// SIMATIC S7-200 SMART project (STEP 7-Micro/WIN SMART), CPU SR40

ORGANIZATION_BLOCK 主程序:OB1
TITLE=程序注释
BEGIN
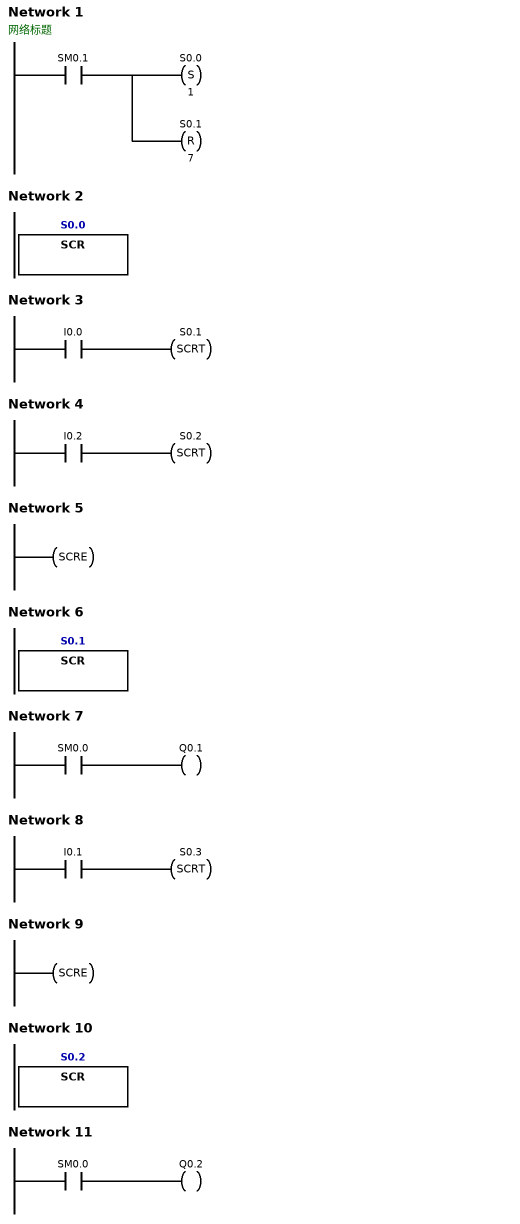
Network 1
// 网络标题
LD     SM0.1
S      S0.0, 1
R      S0.1, 7
Network 2
LSCR   S0.0
Network 3
LD     I0.0
SCRT   S0.1
Network 4
LD     I0.2
SCRT   S0.2
Network 5
SCRE
Network 6
LSCR   S0.1
Network 7
LD     SM0.0
=      Q0.1
Network 8
LD     I0.1
SCRT   S0.3
Network 9
SCRE
Network 10
LSCR   S0.2
Network 11
LD     SM0.0
=      Q0.2
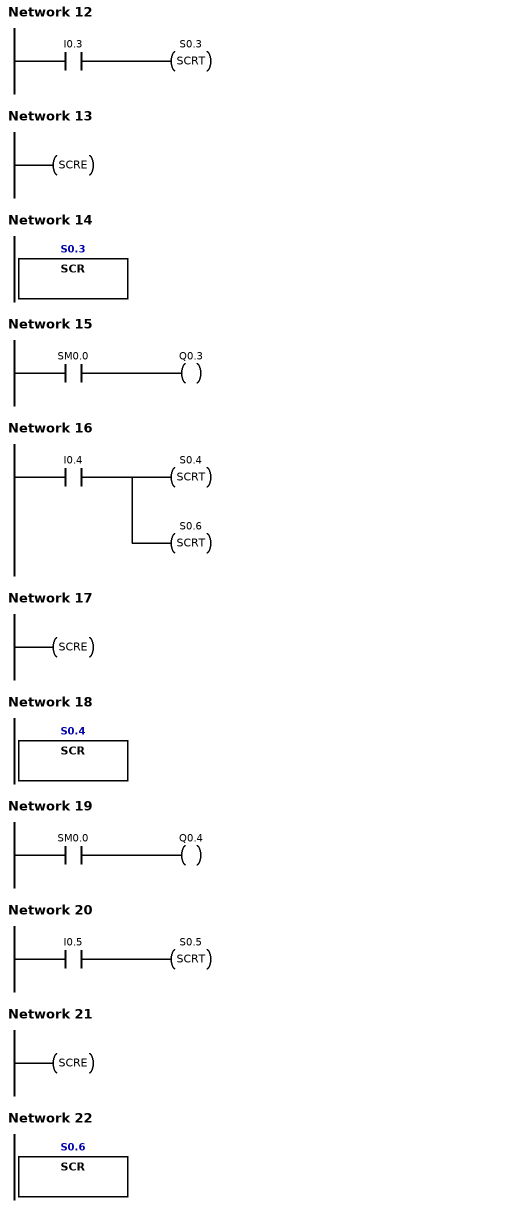
Network 12
LD     I0.3
SCRT   S0.3
Network 13
SCRE
Network 14
LSCR   S0.3
Network 15
LD     SM0.0
=      Q0.3
Network 16
LD     I0.4
SCRT   S0.4
SCRT   S0.6
Network 17
SCRE
Network 18
LSCR   S0.4
Network 19
LD     SM0.0
=      Q0.4
Network 20
LD     I0.5
SCRT   S0.5
Network 21
SCRE
Network 22
LSCR   S0.6
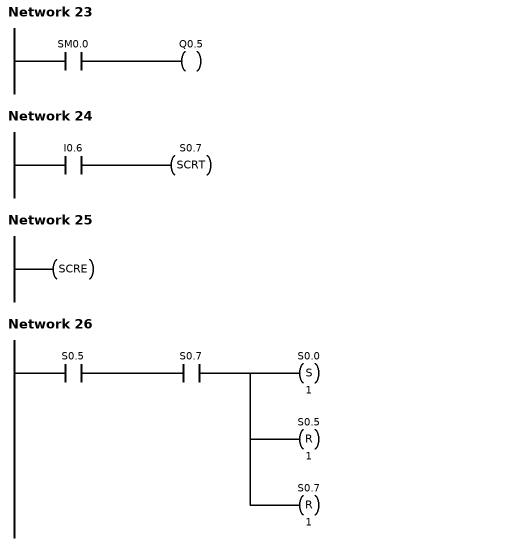
Network 23
LD     SM0.0
=      Q0.5
Network 24
LD     I0.6
SCRT   S0.7
Network 25
SCRE
Network 26
LD     S0.5
A      S0.7
S      S0.0, 1
R      S0.5, 1
R      S0.7, 1
END_ORGANIZATION_BLOCK
